// TIA Portal V19 export
VAR_GLOBAL   // PLC tag table "U2Em3_Output"
   "null(19)" AT %Q171.7 : Bool;   // 备用
   "null(15)" AT %Q170.5 : Bool;   // 备用
   hookClawCylinderWorkPositionU3Em3_2 AT %Q171.0 : Bool;   // U3Em3_Hook claw cylinder 2 working position / Em100_钩爪气缸2工作位
   slideCylinderWorkPositionU3Em3_1 AT %Q170.0 : Bool;   // U3Em3_ Sliding table cylinder 1 working position / Em100_滑台气缸1工作位
   "null(14)" AT %Q170.4 : Bool;   // 备用
   hookClawCylinderHomePositionU3Em3_1 AT %Q170.7 : Bool;   // U3Em3_Hook Claw Cylinder 1 Home Position / Em100_钩爪气缸1原位
   pressureGaugeZeroingU3Em3_1 AT %Q171.4 : Bool;   // U3Em3_Pressure gauge 1 reset to zero / Em100_压力表1清零
   "null(16)" AT %Q171.2 : Bool;   // 备用
   slideCylinderWorkPositionU3Em3_2 AT %Q170.2 : Bool;   // U3Em3_ Sliding table cylinder 2 working position / Em100_滑台气缸2工作位
   pressureGaugeZeroingU3Em3_2 AT %Q171.5 : Bool;   // U3Em3_Pressure gauge 2 reset to zero / Em100_压力表2清零
   slideCylinderHomePositionU3Em3_1 AT %Q170.1 : Bool;   // U3Em3_skid table cylinder 1 original position / Em100_滑台气缸1原位
   hookClawCylinderWorkPositionU3Em3_1 AT %Q170.6 : Bool;   // U3Em3_Hook claw cylinder 1 working position / Em100_钩爪气缸1工作位
   hookClawCylinderHomePositionU3Em3_2 AT %Q171.1 : Bool;   // U3Em3_Hook Claw Cylinder 2 Home Position / Em100_钩爪气缸2原位
   slideCylinderHomePositionU3Em3_2 AT %Q170.3 : Bool;   // U3Em3_skid table cylinder 2 original position / Em100_滑台气缸2原位
   "null(17)" AT %Q171.3 : Bool;   // spare / 备用
   "null(18)" AT %Q171.6 : Bool;   // spare / 备用
END_VAR
